(* CoDeSys 2.3 export: RUN_PRG.EXP *)

(* POU RUN_PRG, CFC *)
PROGRAM RUN_PRG
VAR
	Run: BOOL := TRUE;
	aFS					: ARRAY [0..2] OF FLASHING_SEQUENCE := 	(Colour:=GREEN, Frequency:=0, Relation:=128, NextIndex:=0),
																				(Colour:=RED, Frequency:=0, Relation:=128, NextIndex:=0),
																				(Colour:=ORANGE, Frequency:=0, Relation:=128, NextIndex:=0);
	ptFS				: POINTER TO FLASHING_SEQUENCE;
END_VAR
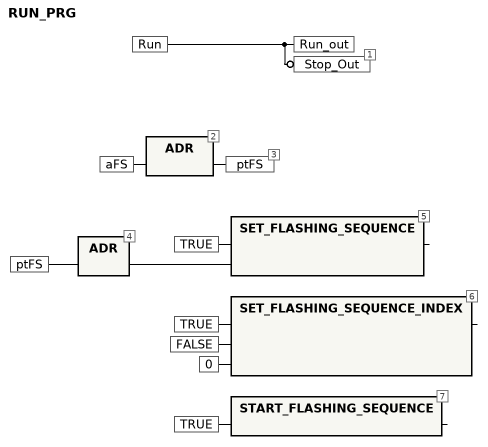
_CFC_ (* Continuous Function Chart, elements in execution order *)
#0 Run_out <= Run
#1 Stop_Out <= NOT Run
#2 ADR(aFS)
#3 ptFS <= #2
#4 ADR(ptFS)
#5 SET_FLASHING_SEQUENCE(TRUE, #4)
#6 SET_FLASHING_SEQUENCE_INDEX(TRUE, FALSE, 0)
#7 START_FLASHING_SEQUENCE(TRUE)
_END_CFC_
(* the same logic as Structured Text *)
Run_out := Run;
Stop_Out := NOT Run;
ptFS := ADR(aFS);
SET_FLASHING_SEQUENCE(TRUE, ADR(ptFS));
SET_FLASHING_SEQUENCE_INDEX(TRUE, FALSE, 0);
START_FLASHING_SEQUENCE(TRUE);
END_PROGRAM
